TYPE (* DataPanel Modules with medium IO density AI Struct + Source Address *)
  (* Version 1.0, 2026-05-28, franz *)
  PACKAGE DataPanel::io::MI::AI;
  IMPORT DataPanel::io::MI::AI::DataPanel_MI_AI::Invalid;
  IMPORT DataPanel::io::MI::const::MI::MI_00;
  DataPanel_MI_AI_S_Dual_SA : STRUCT
    u8SAMember : USINT := MI_00; (* Node SA 224..239 *)
    Up : DataPanel::io::MI::AI::DataPanel_MI_AI_S := Invalid; (* Identify the Port 1A..8B forward, up, right, clockwise *)
    Down : DataPanel::io::MI::AI::DataPanel_MI_AI_S := Invalid; (* Identify the Port 1A..8B backward, down, left, counter-clockwise *)
  END_STRUCT;
END_TYPE
